Universal Robots PolyScope program: PF RRP.urp

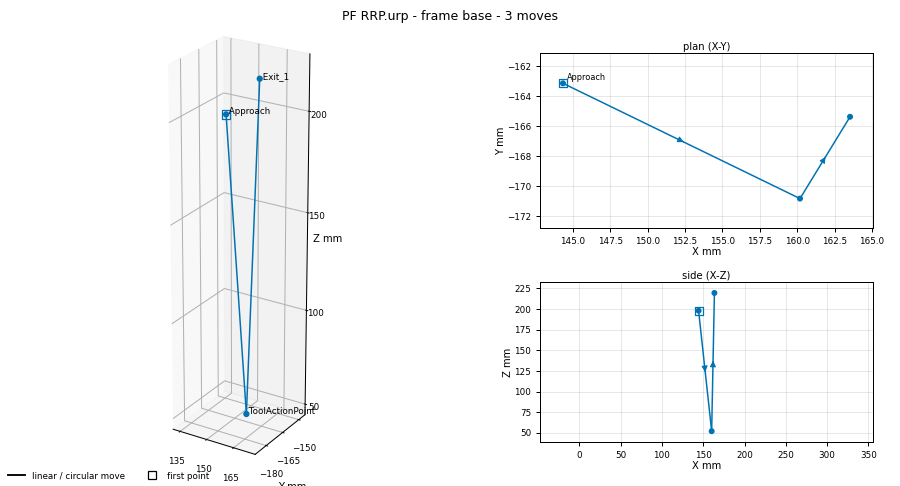
[picture p0: tool path of PF RRP.urp in frame base, 3 of 3 moves have a stored position in this frame; points joined in program order, loops and branches not executed]
Program PF RRP (installation=default directory=/programs createdIn=5.14.5 lastSavedIn=5.14.5 robotSerialNumber=20195300809)
Calibrated DH parameters: a=[-0.000085, -0.20076, -0.212369, 0.000121, -0.000118, 0]; d=[0.15185, -26.306375, 24.753047, 1.684739, 0.085386, 0.092088]; alpha=[1.572149, -0.00522, -0.011864, 1.571339, -1.571085, 0]; deltaTheta=[0, 0.599885, -0.513355, -0.086555, 0.000006, 0]
InitVariablesNode variables(variable(name=Pallet_1_cnt_1, expression=1), variable(name=Pallet_1_lct, expression=1), variable(name=Pallet_1_lno, expression=1), variable(name=Pallet_1_sep, expression=False), variable(name=Pallet_1_tct, expression=1))
Robot Program (runOnlyOnce=false)
  URCap Gripper Activate (Robotiq_Grippers, Robotiq Inc.) dataModel(ResetAndActivateKey=false)
  SafeHome (positionOptionType=SPEED_AND_ACCELERATION speed=1.047198 acceleration=1.396263 nextMotionTime=2)
  URCap Palletizing (polyscope-pallet-impl, Universal Robots) dataModel(palletFeature=Base, isPalletizing=false, rememberTraversal=false, beforeSelected=false, afterSelected=false, Variable(key=referencePoint, variable(featureName=referencePoint)), Variable(key=separatorPoint, variable(featureName=separatorPoint)), Variable(key=name, variable(name=Pallet_1)), Variable(key=layerNumberVariable, variable(name=Pallet_1_lno, initializeExpression=1)), Variable(key=layerCountingVariable, variable(name=Pallet_1_lct, initializeExpression=1)), Variable(key=handleSeparatorVariable, variable(name=Pallet_1_sep, initializeExpression=False)), Variable(key=totalCountVariable, variable(name=Pallet_1_tct, initializeExpression=1)), Length(key=objectHeight value=0.01 unit=M), Variable(key=globalCountingVariable, variable(name=Pallet_1_cnt_1, initializeExpression=1))); state(isChildrenLocked=true)
    URCap Patterns (polyscope-pallet-impl, Universal Robots) state(isChildrenLocked=true)
      URCap Pattern (polyscope-pallet-impl, Universal Robots) dataModel(UUID=0a789ce8-e85e-4730-881f-26af6b7c39b1, patternType=LINE, objects=3, Variable(key=nameVariable, variable(name=Line_Pattern_1))); state(isChildrenLocked=true)
        URCap Item (polyscope-pallet-impl, Universal Robots) dataModel(UUID=3f73535f-4f40-47dc-8fce-d81d1f67adbe, patternType=LINE, index=0, calibrationDeltaTheta=[2.0871938292282843E-8, 0.5998849625986696, -0.513354759222901, -0.08655474087847535, 6.239817607139875E-6, -6.658617090343766E-8], calibrationA=[-8.52060452638757E-5, -0.2007601879611388, -0.2123691625519033, 1.2105607098011576E-4, -1.1833705743435544E-4, 0.0], calibrationD=[0.15184970286177432, -26.306374840159272, 24.75304670983349, 1.6847390881089916, 0.085385969004481, 0.09208826337351553], calibrationAlpha=[1.5721487795181908, -0.005219907129425837, -0.011864150755780208, 1.5713392161993658, -1.5710853432049288, 0.0], calibrationJointChecksum=[-1860213401, -1859864814, -1494669377, -1328152407, -1329437658, -1329056899], calibrationStatus=2, calibrationValidChecksum=true, baseToFeature=[0.0, 0.0, 0.0, 0.0, 0.0, 0.0], TCPOffset=[-3.5417170762830352E-6, -1.6903386905048334E-5, 0.17398062376878348, 7.31767217500838E-5, -3.318045036855908E-5, 5.6030804581462324E-5], Variable(key=variable, variable(name=StartItem_1)), JointPositions(key=jointpositions, JointPosition(key=[1], Angle(key=pos value=-0.173928 unit=RAD)), JointPosition(key=[2], Angle(key=pos value=-1.089065 unit=RAD)), JointPosition(key=[3], Angle(key=pos value=-2.294135 unit=RAD)), JointPosition(key=[4], Angle(key=pos value=-1.299985 unit=RAD)), JointPosition(key=[5], Angle(key=pos value=1.52529 unit=RAD)), JointPosition(key=[6], Angle(key=pos value=-0.207832 unit=RAD))))
        URCap Item (polyscope-pallet-impl, Universal Robots) dataModel(UUID=fe91c25c-b58f-4ec5-bbe5-a7f152dd7ebb, patternType=LINE, index=1, calibrationDeltaTheta=[2.0871938292282843E-8, 0.5998849625986696, -0.513354759222901, -0.08655474087847535, 6.239817607139875E-6, -6.658617090343766E-8], calibrationA=[-8.52060452638757E-5, -0.2007601879611388, -0.2123691625519033, 1.2105607098011576E-4, -1.1833705743435544E-4, 0.0], calibrationD=[0.15184970286177432, -26.306374840159272, 24.75304670983349, 1.6847390881089916, 0.085385969004481, 0.09208826337351553], calibrationAlpha=[1.5721487795181908, -0.005219907129425837, -0.011864150755780208, 1.5713392161993658, -1.5710853432049288, 0.0], calibrationJointChecksum=[-1860213401, -1859864814, -1494669377, -1328152407, -1329437658, -1329056899], calibrationStatus=2, calibrationValidChecksum=true, baseToFeature=[0.0, 0.0, 0.0, 0.0, 0.0, 0.0], TCPOffset=[1.0071926361848726E-5, 8.602880394725787E-7, 0.1739852719267095, 2.0855834250884404E-5, 6.795005034418234E-7, 3.080959374802387E-5], Variable(key=variable, variable(name=EndItem_1)), JointPositions(key=jointpositions, JointPosition(key=[1], Angle(key=pos value=-0.092552 unit=RAD)), JointPosition(key=[2], Angle(key=pos value=-1.956869 unit=RAD)), JointPosition(key=[3], Angle(key=pos value=-1.469857 unit=RAD)), JointPosition(key=[4], Angle(key=pos value=-1.231764 unit=RAD)), JointPosition(key=[5], Angle(key=pos value=1.550912 unit=RAD)), JointPosition(key=[6], Angle(key=pos value=-0.09466 unit=RAD))))
    URCap Layers (polyscope-pallet-impl, Universal Robots) dataModel(separators=[false], selectedPatterns=[0a789ce8-e85e-4730-881f-26af6b7c39b1])
    URCap At Each Item (polyscope-pallet-impl, Universal Robots) dataModel(selectedPattern=0a789ce8-e85e-4730-881f-26af6b7c39b1, selectedPosition=3f73535f-4f40-47dc-8fce-d81d1f67adbe, Approach_calibrationDeltaTheta=[2.0871938292282843E-8, 0.5998849625986696, -0.513354759222901, -0.08655474087847535, 6.239817607139875E-6, -6.658617090343766E-8], Approach_calibrationA=[-8.52060452638757E-5, -0.2007601879611388, -0.2123691625519033, 1.2105607098011576E-4, -1.1833705743435544E-4, 0.0], Approach_calibrationD=[0.15184970286177432, -26.306374840159272, 24.75304670983349, 1.6847390881089916, 0.085385969004481, 0.09208826337351553], Approach_calibrationAlpha=[1.5721487795181908, -0.005219907129425837, -0.011864150755780208, 1.5713392161993658, -1.5710853432049288, 0.0], Approach_calibrationJointChecksum=[-1860213401, -1859864814, -1494669377, -1328152407, -1329437658, -1329056899], Approach_calibrationStatus=2, Approach_calibrationValidChecksum=true, Approach_baseToFeature=[0.0, 0.0, 0.0, 0.0, 0.0, 0.0], Approach_TCPOffset=[1.4220217284810488E-6, -2.2608274058893985E-5, 0.17399111092200326, 6.484771814642449E-5, 3.587997059201472E-5, -8.862925324860848E-5], Exit_calibrationDeltaTheta=[2.0871938292282843E-8, 0.5998849625986696, -0.513354759222901, -0.08655474087847535, 6.239817607139875E-6, -6.658617090343766E-8], Exit_calibrationA=[-8.52060452638757E-5, -0.2007601879611388, -0.2123691625519033, 1.2105607098011576E-4, -1.1833705743435544E-4, 0.0], Exit_calibrationD=[0.15184970286177432, -26.306374840159272, 24.75304670983349, 1.6847390881089916, 0.085385969004481, 0.09208826337351553], Exit_calibrationAlpha=[1.5721487795181908, -0.005219907129425837, -0.011864150755780208, 1.5713392161993658, -1.5710853432049288, 0.0], Exit_calibrationJointChecksum=[-1860213401, -1859864814, -1494669377, -1328152407, -1329437658, -1329056899], Exit_calibrationStatus=2, Exit_calibrationValidChecksum=true, Exit_baseToFeature=[0.0, 0.0, 0.0, 0.0, 0.0, 0.0], Exit_TCPOffset=[7.191351677565683E-6, 1.6397458372507945E-6, 0.1739935690312755, 2.474130948248851E-6, 3.8466636449150564E-5, 1.1868100585119471E-5], currentWizardState=MANUAL, Pose(key=refBaseToFeature, Position(key=posePosition, Length(key=X value=0 unit=M), Length(key=Y value=0 unit=M), Length(key=Z value=0 unit=M)), Rotation(key=poseRotation, Angle(key=RX value=0 unit=RAD), Angle(key=RY value=0 unit=RAD), Angle(key=RZ value=0 unit=RAD))), Pose(key=refPose, Position(key=posePosition, Length(key=X value=0.160185 unit=M), Length(key=Y value=-0.170831 unit=M), Length(key=Z value=0.052109 unit=M)), Rotation(key=poseRotation, Angle(key=RX value=2.2482 unit=RAD), Angle(key=RY value=-2.172551 unit=RAD), Angle(key=RZ value=0.069903 unit=RAD))), JointPositions(key=Approach_jointpositions, JointPosition(key=[1], Angle(key=pos value=-0.173923 unit=RAD)), JointPosition(key=[2], Angle(key=pos value=-1.069634 unit=RAD)), JointPosition(key=[3], Angle(key=pos value=-1.6043 unit=RAD)), JointPosition(key=[4], Angle(key=pos value=-1.998509 unit=RAD)), JointPosition(key=[5], Angle(key=pos value=1.540701 unit=RAD)), JointPosition(key=[6], Angle(key=pos value=-0.182381 unit=RAD))), JointPositions(key=Exit_jointpositions, JointPosition(key=[1], Angle(key=pos value=-0.169081 unit=RAD)), JointPosition(key=[2], Angle(key=pos value=-1.245768 unit=RAD)), JointPosition(key=[3], Angle(key=pos value=-1.377631 unit=RAD)), JointPosition(key=[4], Angle(key=pos value=-2.107994 unit=RAD)), JointPosition(key=[5], Angle(key=pos value=1.540976 unit=RAD)), JointPosition(key=[6], Angle(key=pos value=-0.143775 unit=RAD))))
      URCap Generated Movements (polyscope-pallet-impl, Universal Robots) state(isChildrenLocked=true)
        MoveJ speed 60 deg/s, acceleration 80 deg/s^2 (useActiveTCP=true) feature=referencePoint
          Waypoint Approach: TCP in base x=144.347 y=-163.129 z=198.095 mm, rx=-2.237 ry=2.1994 rz=-0.072 rad; joints [-9.965, -61.285, -91.92, -114.506, 88.276, -10.45] deg; TCP offset x=0.001 y=-0.023 z=173.991 mm, rx=0.0001 ry=0 rz=-0.0001 rad; feature pose in base x=160.185 y=-170.831 z=52.109 mm, rx=2.2482 ry=-2.1726 rz=0.0699 rad
        MoveL speed 250 mm/s, acceleration 1200 mm/s^2 (useActiveTCP=true) feature(featureName=referencePoint)
          Waypoint ToolActionPoint: TCP in base x=160.185 y=-170.831 z=52.109 mm, rx=2.2482 ry=-2.1726 rz=0.0699 rad; joints [-9.965, -62.399, -131.444, -74.484, 87.393, -11.908] deg; TCP offset x=-0.004 y=-0.017 z=173.981 mm, rx=0.0001 ry=0 rz=0.0001 rad
        Folder Tool action
          URCap Gripper (Robotiq_Grippers, Robotiq Inc.) dataModel(position=100.0, force=0.0, speed=0.0, positionInDouble=100.0, forceInDouble=0.0, speedInDouble=0.0, slaveIds=[9], blocking=true)
        MoveL speed 250 mm/s, acceleration 1200 mm/s^2 (useActiveTCP=true) feature(featureName=referencePoint)
          Waypoint Exit_1: TCP in base x=163.529 y=-165.366 z=219.542 mm, rx=2.1843 ry=-2.2163 rz=-0.0031 rad; joints [-9.688, -71.377, -78.932, -120.779, 88.291, -8.238] deg; TCP offset x=0.007 y=0.002 z=173.994 mm, rx=0 ry=0 rz=0 rad
